FUNCTION_BLOCK T_AddComponentAddedToList EXTENDS T_UnitTestBase
VAR
  list : T_ComponentsCollection;
  newComponent : T_ComponentMock;
  result : BOOL;
END_VAR

result := list.AddComponent(newComponent);

assertion.AssertEquals_BOOL(TRUE, result, 'list.AddComponent(newComponent);');
TestFinished();

END_FUNCTION_BLOCK

(* stored: Version 1.1.0.1, ProductVersion 3.1.4024.12
   POU T_AddComponentAddedToList: Id {0a8b6a35-5a1f-409c-9210-a2cfd61be5f4}, SpecialFunc None *)
